# B&R Automation Studio project lab1
Automation Studio 4.5.2.102

## Configuration Config1

CPU 4PP065.0351-X74, AutomationRuntime D4.52, Build 4.1.2, Vc V4.52.0

### Task classes (Cpu.sw)
```
Cyclic#4:
  Program <- Program.prg
Libraries: Library
```

### Hardware
```
4PP065_0351_X74 : 4PP065.0351-X74 v1.0.7.0
  Connector IF5:
    ActivateDevice = 1
  ConfigurationID = lab1_Config1
  Simulation = 1
  KeyMappingFile = VC\4PP065_0351_X74.dis
```

## Logical view

Binary libraries used (declarations not repeated): operator, runtime, astime, AsIecCon

### Package Logical/Libraries - Global libraries

### Library Logical/Libraries/Library (ANSIC)

#### Library.fun - Exported functions and function blocks
```iecst
{REDUND_ERROR} FUNCTION_BLOCK FB_integrator (*TODO: Add your comment here*) (*$GROUP=User,$CAT=User,$GROUPICON=User.png,$CATICON=User.png*)
	VAR_INPUT
		in : {REDUND_UNREPLICABLE} REAL;
	END_VAR
	VAR_OUTPUT
		out : {REDUND_UNREPLICABLE} REAL;
	END_VAR
	VAR
		dt : {REDUND_UNREPLICABLE} REAL;
		prev_value : REAL;
	END_VAR
END_FUNCTION_BLOCK

{REDUND_ERROR} {REDUND_UNREPLICABLE} FUNCTION_BLOCK FB_motor (*TODO: Add your comment here*) (*$GROUP=User,$CAT=User,$GROUPICON=User.png,$CATICON=User.png*)
	VAR_INPUT
		u : {REDUND_UNREPLICABLE} REAL;
	END_VAR
	VAR_OUTPUT
		w : {REDUND_UNREPLICABLE} REAL;
		phi : {REDUND_UNREPLICABLE} REAL;
	END_VAR
	VAR
		integrator : {REDUND_UNREPLICABLE} FB_integrator;
		T_m : {REDUND_UNREPLICABLE} REAL;
		k_e : {REDUND_UNREPLICABLE} REAL;
		dt : {REDUND_UNREPLICABLE} REAL;
	END_VAR
END_FUNCTION_BLOCK

{REDUND_ERROR} FUNCTION_BLOCK FB_controller (*TODO: Add your comment here*) (*$GROUP=User,$CAT=User,$GROUPICON=User.png,$CATICON=User.png*)
	VAR_INPUT
		e : {REDUND_UNREPLICABLE} REAL;
	END_VAR
	VAR_OUTPUT
		u : {REDUND_UNREPLICABLE} REAL;
	END_VAR
	VAR
		k_p : {REDUND_UNREPLICABLE} REAL;
		k_i : {REDUND_UNREPLICABLE} REAL;
		integrator : {REDUND_UNREPLICABLE} FB_integrator;
		iyOld : {REDUND_UNREPLICABLE} REAL;
		max_abs_value : {REDUND_UNREPLICABLE} REAL;
		dt : {REDUND_UNREPLICABLE} REAL;
		last_sum : REAL;
	END_VAR
END_FUNCTION_BLOCK
```

#### FB_integrator.c
```c
#include <bur/plctypes.h>
#ifdef __cplusplus
	extern "C"
	{
#endif
	#include "Library.h"
#ifdef __cplusplus
	};
#endif
/* TODO: Add your comment here */
void FB_integrator(struct FB_integrator* inst)
{
	/*TODO: Add your code here*/
	inst->out = inst->dt * inst->in + inst->out;
	inst->prev_value = inst->out;
}
```

#### FB_motor.c
```c
#include <bur/plctypes.h>
#ifdef __cplusplus
	extern "C"
	{
#endif
	#include "Library.h"
#ifdef __cplusplus
	};
#endif
/* TODO: Add your comment here */
void FB_motor(struct FB_motor* inst)
{
	/*TODO: Add your code here*/
	REAL a = inst->u / inst->k_e - inst->w;
	REAL b = a / inst->T_m;

	inst->integrator.in = b;
	FB_integrator(&inst->integrator);

	inst->w = inst->integrator.out;

}
```

#### FB_controller.c
```c
#include <bur/plctypes.h>
#ifdef __cplusplus
	extern "C"
	{
#endif
	#include "Library.h"
#ifdef __cplusplus
	};
#endif
/* TODO: Add your comment here */
void FB_controller(struct FB_controller* inst)
{
	/*TODO: Add your code here*/
	REAL a = inst->e * inst->k_p;
	REAL b = inst->e * inst->k_i; // * inst-> dt;

	a = a > inst->max_abs_value ? inst->max_abs_value : a;
	a = a < -inst->max_abs_value ? -inst->max_abs_value : a;

	inst->integrator.in = b + inst->iyOld;
	FB_integrator(&inst->integrator);

	REAL sum = a + inst->integrator.out;

	inst->u = sum;
	inst->u = inst->u > inst->max_abs_value ? inst->max_abs_value : inst->u;
	inst->u = inst->u < -inst->max_abs_value ? -inst->max_abs_value : inst->u;

	inst->iyOld = inst->u - sum;

}
```

### Program Logical/Program (ANSIC)

#### Variables.var
```iecst
VAR
	fb_motor : FB_motor;
	fb_controller : FB_controller;
	counter : UINT;
	speed : REAL;
	enable : BOOL;
	fb_motor1 : FB_motor;
	fb_motor2 : FB_motor;
END_VAR
```

#### Main.c
```c
#include <bur/plctypes.h>

#ifdef _DEFAULT_INCLUDES
	#include <AsDefault.h>
#endif

void _INIT ProgramInit(void)
{
	fb_motor.dt = 0.01;
	fb_motor.k_e = 0.24;
	fb_motor.T_m = 0.03;
	fb_motor.u = 0;
	fb_motor.integrator.dt = 0.01;

	fb_motor2.dt = 0.01;
	fb_motor2.k_e = 0.24;
	fb_motor2.T_m = 0.03;
	fb_motor2.u = 0;
	fb_motor2.integrator.dt = 0.01;

	fb_controller.dt = 0.01;
	fb_controller.integrator.dt = 0.01;
	fb_controller.k_i = 24;
	fb_controller.k_p = 0.24*3;
	fb_controller.max_abs_value = 24.0;

	speed = 0;
	counter = 0;
	enable=1;

}

void _CYCLIC ProgramCyclic(void)
{
	if (enable)
	{
		if (counter == 100)
		{
			speed = 50;
		}
		else if (counter == 250)
		{
			speed = 0;
			counter = 0;
		}
		counter++;

		fb_controller.e = speed - fb_motor.w;
		FB_controller(&fb_controller);

		fb_motor.u = fb_controller.u;

		fb_motor2.u = speed * fb_motor2.k_e;

		FB_motor(&fb_motor);
		FB_motor(&fb_motor2);

	}
}

void _EXIT ProgramExit(void)
{

}
```

Listed in the project but not available here: Logical/Global.typ, Logical/Global.var, Logical/Libraries/Library/Types.typ, Logical/Libraries/Library/Constants.var
